// TIA Portal project "HMI_Tank_Filling" (V17)

(* hardware
DEVICE "HMI_1"  KTP700 Basic PN
   slot 0: "HMI_1"  KTP700 Basic PN  6AV2 123-2GB03-0AX0  17.0.0.0
   slot 1: "HMI_RT_1"  KTP700 Basic PN  6AV2 123-2GB03-0AX0  17.0.0.0
   slot 5: "HMI_1.IE_CP_1"  PROFINET Interface  17.0.0.0
      slot 1: "PROFINET Interface_1"  PROFINET Interface
         slot 1: "Port_1"  Port
DEVICE "S7-1200 station_1"  S7-1200 Station
   slot 0: "Rack_0"  S7-1200 Rack  Rack  V1.0
   slot 1: "PLC_1"  CPU 1215C DC/DC/DC  6ES7 215-1AG40-0XB0  V4.5
   slot 2: "AQ 2x14BIT_1"  SM 1232 AQ2  6ES7 232-4HB32-0XB0  V2.1
*)

// ===== PLC "PLC_1"  CPU 1215C DC/DC/DC =====

VAR_GLOBAL   // PLC tag table "Default tag table"
   "valve_filling" AT %QW30 : Int;
   "HMI_Switch" AT %M10.0 : Bool;
   "valve_unloading" AT %QW32 : Int;
   "level_detection_sensor" AT %IW30 : Int;
   "Tag_1" AT %MD20 : DWord;
   "water_level" AT %MD24 : Real;
   "HMI_water_level" AT %MW30 : Int;
END_VAR

ORGANIZATION_BLOCK "Main"   // OB1, LAD, ProgramCycle
TITLE = "Main Program Sweep (Cycle)"
{ S7_Optimized_Access := 'TRUE' }
VERSION : 0.1
   VAR_INPUT
      Initial_Call : Bool;   // Initial call of this OB
      Remanence : Bool;   // =True, if remanent data are available
   END_VAR
BEGIN

REGION Network 1
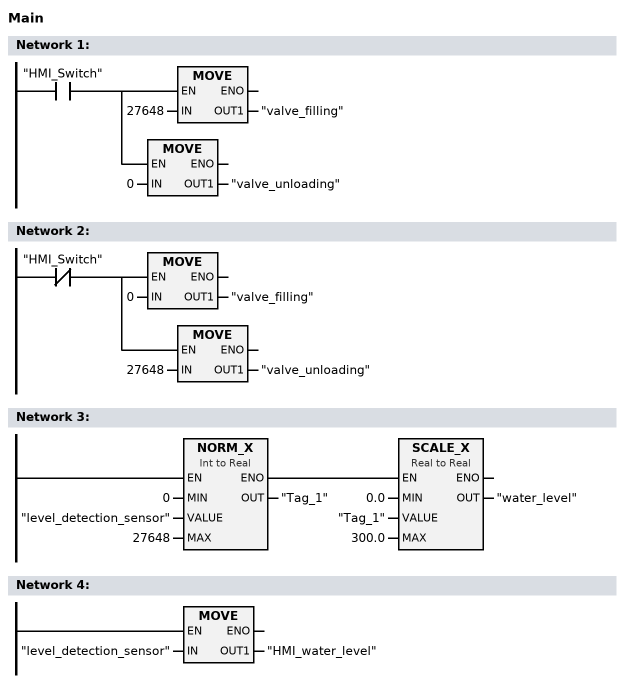
   RUNG wire#powerrail
      Contact( "HMI_Switch" )
      wire#w1
      Move(in := 27648, out1 => "valve_filling")
   END_RUNG
   RUNG wire#w1
      Move(in := 0, out1 => "valve_unloading")
   END_RUNG
   // the same network as SCL:
   IF "HMI_Switch" THEN
       "valve_filling" := 27648;
       "valve_unloading" := 0;
   END_IF;
END_REGION

REGION Network 2
   RUNG wire#powerrail
      I_Contact( "HMI_Switch" )
      wire#w1
      Move(in := 0, out1 => "valve_filling")
   END_RUNG
   RUNG wire#w1
      Move(in := 27648, out1 => "valve_unloading")
   END_RUNG
   // the same network as SCL:
   IF NOT "HMI_Switch" THEN
       "valve_filling" := 0;
       "valve_unloading" := 27648;
   END_IF;
END_REGION

REGION Network 3
   RUNG wire#powerrail
      { S7_Templates := "[SrcType := Int, DestType := Real]" } Normalize(min := 0, value := "level_detection_sensor", max := 27648, out => "Tag_1")
      { S7_Templates := "[SrcType := Real, DestType := Real]" } Scale(min := 0.0, value := "Tag_1", max := 300.0, out => "water_level")
   END_RUNG
   // the same network as SCL:
   "Tag_1" := NORM_X(MIN := 0, VALUE := "level_detection_sensor", MAX := 27648);
   "water_level" := SCALE_X(MIN := 0.0, VALUE := "Tag_1", MAX := 300.0);
END_REGION

REGION Network 4
   RUNG wire#powerrail
      Move(in := "level_detection_sensor", out1 => "HMI_water_level")
   END_RUNG
   // the same network as SCL:
   "HMI_water_level" := "level_detection_sensor";
END_REGION
END_ORGANIZATION_BLOCK

(* ===== HMI "HMI_RT_1" =====
system functions are stored by id; their names below are inferred from use
connection "HMI_Connection_1": ETHERNET, SMART_S7_1200_OMS

HMI tags "Default tag table"
   "Tag_ScreenNumber" : UInt, internal
   "HMI_Switch" : Bool = PLC HMI_Switch AT %M10.0, 1 s
   "water_level" : Real = PLC water_level AT %MD24, 1 s
   "HMI_water_level" : Int = PLC HMI_water_level AT %MW30, 1 s

screen "Root screen" 800x480
   on GenerateScreen: SetTag("Tag_ScreenNumber", 1)
   TextField "Text field_1" at 321,14 size 161x32; Text 'WATER TANK'
   Switch "Switch_1" at 305,418 size 193x37; CaptionText 'Switch'; TextOff 'FILL THE TANK'; TextOn 'UNLOAD THE TANK'
      ProcessValue <- "HMI_Switch"
   Bar "Bar_1" at 363,60 size 80x338; MinimumValue 0; MaximumValue 300
      ProcessValue <- "water_level"
   IOField "I/O field_1" at 498,206 size 96x32; FormatPattern 999
      ProcessValue <- "HMI_water_level"
   TextField "Text field_2" at 602,211 size 120x23; Text 'WATER LEVEL'
*)